Staubli VAL3: getFunctionSel.pgx

public program getFunctionSel(string& x_sName[])
  local string l_sMessage
begin
  //
  // define your message for the
  // function KEY
  //
  // NOTE is an ARRAY[0..7]
  //
  // example:
  // x_sName[1]="DEMO"
  // active the F2 button
  //
  // Set Home Program
  call language:message(l_sMessage,135)
  x_sName[2]=l_sMessage
  call language:message(l_sMessage,136)
  x_sName[3]=l_sMessage
end
